TEXTLIST TextList_02
  0 = 'Czy napewno usunąć recepturę ?' | pl: 'Czy napewno usunąć recepturę ?' | en: 'Are you sure you want to delete the recipe?' | de: 'Möchten Sie das Rezept wirklich löschen?'
   = ''
END_TEXTLIST

(* stored: Version 1.1.0.1
   TextList TextList_02: Id {71a36f57-212e-074a-249a-1cb71d504b6c} *)
